(* CoDeSys 2.3 export: PARAMETERGROUP_TS.EXP *)

(* Data type in Diag/Parameter *)
TYPE ParameterGroup_ts :
STRUCT
	GroupName_as8			: STRING(32);
(*	GroupName_as8			: ARRAY [1..4] OF STRING(32);*)
	Param_as					: ARRAY [1..8] OF Parameter_ts;
END_STRUCT
END_TYPE
